//
// In order for extender of this FB
// -- to set specific logger name category call SetLoggerCategoryName(<the name>) (from FB_Init())

FUNCTION_BLOCK FB_BaseFb
VAR
	{attribute 'OPC.UA.DA' := '0'}
	LogMsg_0: LogMsg;
	{attribute 'OPC.UA.DA' := '0'}
	pLogMsgToUse: POINTER TO LogMsg := ADR(LogMsg_0);
	{attribute 'OPC.UA.DA' := '0'}
	DINT_0 :DINT;
	
END_VAR

METHOD FB_init : BOOL
VAR_INPUT
	bInitRetains : BOOL; // if TRUE, the retain variables are initialized (warm start / cold start)
	bInCopyCode : BOOL;  // if TRUE, the instance afterwards gets moved into the copy code (online change)
END_VAR
END_METHOD

METHOD PUBLIC GetLoggerCategoryName : pointer to string
VAR_INPUT
END_VAR
GetLoggerCategoryName	:= ADR(THIS^.pLogMsgToUse^.logData.category);
END_METHOD

METHOD LogError
VAR_INPUT
	textMessage : STRING[LOG_MSG_TEXT_LENGTH];
	param1 : DINT;
	param2 : DINT;
	param3 : DINT;	
	param4 : DINT;
	param5 : DINT;
	param6 : DINT;	
END_VAR
pLogMsgToUse^.LogMsg(LOG_ERROR, textMessage, param1, param2, param3, param4, param5, param6);
LogTransfer();
END_METHOD

METHOD LogError_v2 : BOOL
VAR_INPUT
	textMessage : STRING[LOG_MSG_TEXT_LENGTH];
	param1 : ANY;
	param2 : ANY;
	param3 : ANY;	
	param4 : ANY;
	param5 : ANY;
	param6 : ANY;	
	param7 : ANY;	
	param8 : ANY;
	param9 : ANY;
	param10 : ANY;		
END_VAR
VAR
	param1_Arg   :T_arg;
	param2_Arg   :T_arg;
	param3_Arg   :T_arg;
	param4_Arg   :T_arg;
	param5_Arg   :T_arg;
	param6_Arg   :T_arg;
	param7_Arg   :T_arg;
	param8_Arg   :T_arg;
	param9_Arg   :T_arg;
	param10_Arg  :T_arg;
END_VAR

param1_Arg	:=fnCnvToTarg(param1);
param2_Arg	:=fnCnvToTarg(param2);
param3_Arg	:=fnCnvToTarg(param3);
param4_Arg	:=fnCnvToTarg(param4);
param5_Arg	:=fnCnvToTarg(param5);
param6_Arg	:=fnCnvToTarg(param6);
param7_Arg	:=fnCnvToTarg(param7);
param8_Arg	:=fnCnvToTarg(param8);
param9_Arg	:=fnCnvToTarg(param9);
param10_Arg	:=fnCnvToTarg(param10);

pLogMsgToUse^.LogMsg_v2(LOG_ERROR, textMessage, param1_Arg, param2_Arg, param3_Arg, param4_Arg, param5_Arg, param6_Arg, param7_Arg ,param8_Arg ,param9_Arg,param10_Arg);
LogTransfer();
END_METHOD

METHOD LogInfo
VAR_INPUT
	textMessage : STRING[LOG_MSG_TEXT_LENGTH];
	param1 : DINT;
	param2 : DINT;
	param3 : DINT;	
	param4 : DINT;
	param5 : DINT;
	param6 : DINT;	
END_VAR
pLogMsgToUse^.LogMsg(LOG_INFO, textMessage, param1, param2, param3, param4, param5, param6);
LogTransfer();
END_METHOD

METHOD LogInfo_v2 : BOOL
VAR_INPUT
	textMessage : STRING[LOG_MSG_TEXT_LENGTH];
	param1 : ANY;
	param2 : ANY;
	param3 : ANY;	
	param4 : ANY;
	param5 : ANY;
	param6 : ANY;	
	param7 : ANY;	
	param8 : ANY;
	param9 : ANY;
	param10 : ANY;		
END_VAR
VAR
	param1_Arg   :T_arg;
	param2_Arg   :T_arg;
	param3_Arg   :T_arg;
	param4_Arg   :T_arg;
	param5_Arg   :T_arg;
	param6_Arg   :T_arg;
	param7_Arg   :T_arg;
	param8_Arg   :T_arg;
	param9_Arg   :T_arg;
	param10_Arg  :T_arg;
END_VAR

param1_Arg	:=fnCnvToTarg(param1);
param2_Arg	:=fnCnvToTarg(param2);
param3_Arg	:=fnCnvToTarg(param3);
param4_Arg	:=fnCnvToTarg(param4);
param5_Arg	:=fnCnvToTarg(param5);
param6_Arg	:=fnCnvToTarg(param6);
param7_Arg	:=fnCnvToTarg(param7);
param8_Arg	:=fnCnvToTarg(param8);
param9_Arg	:=fnCnvToTarg(param9);
param10_Arg	:=fnCnvToTarg(param10);

pLogMsgToUse^.LogMsg_v2(LOG_INFO, textMessage, param1_Arg, param2_Arg, param3_Arg, param4_Arg, param5_Arg, param6_Arg, param7_Arg ,param8_Arg ,param9_Arg,param10_Arg);
LogTransfer();
END_METHOD

METHOD LogTransfer
fnLogTransfer(pLogMsgToUse);
END_METHOD

METHOD LogWarning
VAR_INPUT
	textMessage : STRING[LOG_MSG_TEXT_LENGTH];
	param1 : DINT;
	param2 : DINT;
	param3 : DINT;	
	param4 : DINT;
	param5 : DINT;
	param6 : DINT;	
END_VAR
pLogMsgToUse^.LogMsg(LOG_WARNING, textMessage, param1, param2, param3, param4, param5, param6);
LogTransfer();
END_METHOD

METHOD LogWarning_v2 : BOOL
VAR_INPUT
	textMessage : STRING[LOG_MSG_TEXT_LENGTH];
	param1 : ANY;
	param2 : ANY;
	param3 : ANY;	
	param4 : ANY;
	param5 : ANY;
	param6 : ANY;	
	param7 : ANY;	
	param8 : ANY;
	param9 : ANY;
	param10 : ANY;		
END_VAR
VAR
	param1_Arg   :T_arg;
	param2_Arg   :T_arg;
	param3_Arg   :T_arg;
	param4_Arg   :T_arg;
	param5_Arg   :T_arg;
	param6_Arg   :T_arg;
	param7_Arg   :T_arg;
	param8_Arg   :T_arg;
	param9_Arg   :T_arg;
	param10_Arg  :T_arg;
END_VAR

param1_Arg	:=fnCnvToTarg(param1);
param2_Arg	:=fnCnvToTarg(param2);
param3_Arg	:=fnCnvToTarg(param3);
param4_Arg	:=fnCnvToTarg(param4);
param5_Arg	:=fnCnvToTarg(param5);
param6_Arg	:=fnCnvToTarg(param6);
param7_Arg	:=fnCnvToTarg(param7);
param8_Arg	:=fnCnvToTarg(param8);
param9_Arg	:=fnCnvToTarg(param9);
param10_Arg	:=fnCnvToTarg(param10);

pLogMsgToUse^.LogMsg_v2(LOG_WARNING, textMessage, param1_Arg, param2_Arg, param3_Arg, param4_Arg, param5_Arg, param6_Arg, param7_Arg ,param8_Arg ,param9_Arg,param10_Arg);
LogTransfer();
END_METHOD

METHOD SetLogger
VAR_INPUT
	logMsgToUse: REFERENCE TO LogMsg;
END_VAR
IF(__ISVALIDREF(logMsgToUse)) THEN
	pLogMsgToUse := ADR(logMsgToUse);
END_IF
END_METHOD

METHOD SetLoggerCategoryName
VAR_INPUT
	categoryName: STRING;	// Removed "REFERENCE TO "
END_VAR
categoryName[LOG_MSG_CATEGORY_LENGTH - 1] := 0;

// do not use pLogMsgToUse since the external logger logger could has be set
LogMsg_0.InitLogger(categoryName, 0,0);
END_METHOD

END_FUNCTION_BLOCK

(* stored: Version 1.1.0.1, ProductVersion 3.1.4024.3
   POU FB_BaseFb: Id {20615775-f709-0a1a-3148-c70fff74a325}, SpecialFunc None
   Method FB_init: Id {9656bbc2-4143-0898-31c3-0a70089a4b13}
   Method GetLoggerCategoryName: Id {dca232f9-6d2b-4000-85e7-8133841261dc}
   Method LogError: Id {1d9eb8c5-b473-0e26-3ef6-2c31823bc364}
   Method LogError_v2: Id {560912c7-ebac-4276-b060-d60c6024e8ac}
   Method LogInfo: Id {e021add1-9af5-0417-15fb-e48ba4956979}
   Method LogInfo_v2: Id {e2599e53-39c4-48a6-a424-2bb54be4856c}
   Method LogTransfer: Id {da0ee736-797e-046e-1d99-9d96cc97d542}
   Method LogWarning: Id {f4ec3c90-7894-06ff-1ee8-70db9ba16242}
   Method LogWarning_v2: Id {bf168128-2a82-4368-8877-14c1e708d5e3}
   Method SetLogger: Id {499c98e5-0ca0-0320-095d-6664e9beb2c2}
   Method SetLoggerCategoryName: Id {aaaf4ea5-eb37-0aa3-2519-f60aae6b54ca} *)
